TYPE ST_AbsorptionChillerDefaultParameters :
STRUCT
	aSetPointLimitsTemperature : ARRAY[1..2] OF REAL := [10,30];
END_STRUCT
END_TYPE

(* stored: Version 1.1.0.1, ProductVersion 3.1.4024.10
   DUT ST_AbsorptionChillerDefaultParameters: Id {d6734cbc-2bed-4785-93a6-f9f7f511b043} *)
